SUBAPPLICATION Uebung_087a1 (* Beispiel für E_DEMUX_4 *)
  (* Standard: 61499-2; Description: Copyright (c) 2023 Meisterschulen am Ostbahnhof This program and the accompanying materials are made available under the terms of the Eclipse Public License 2.0 which is available at https://www.eclipse.org/legal/epl-2.0/ SPDX-License-Identifier: EPL-2.0 Beispiel für E_CTD Aufwärts zählen UAO Curriculum Module 3 - The IEC 61499 Standard, Seite 93 *)
  (* Version 1.0, 2023-10-23, Franz Höpfinger, Meisterschulen am Ostbahnhof *)
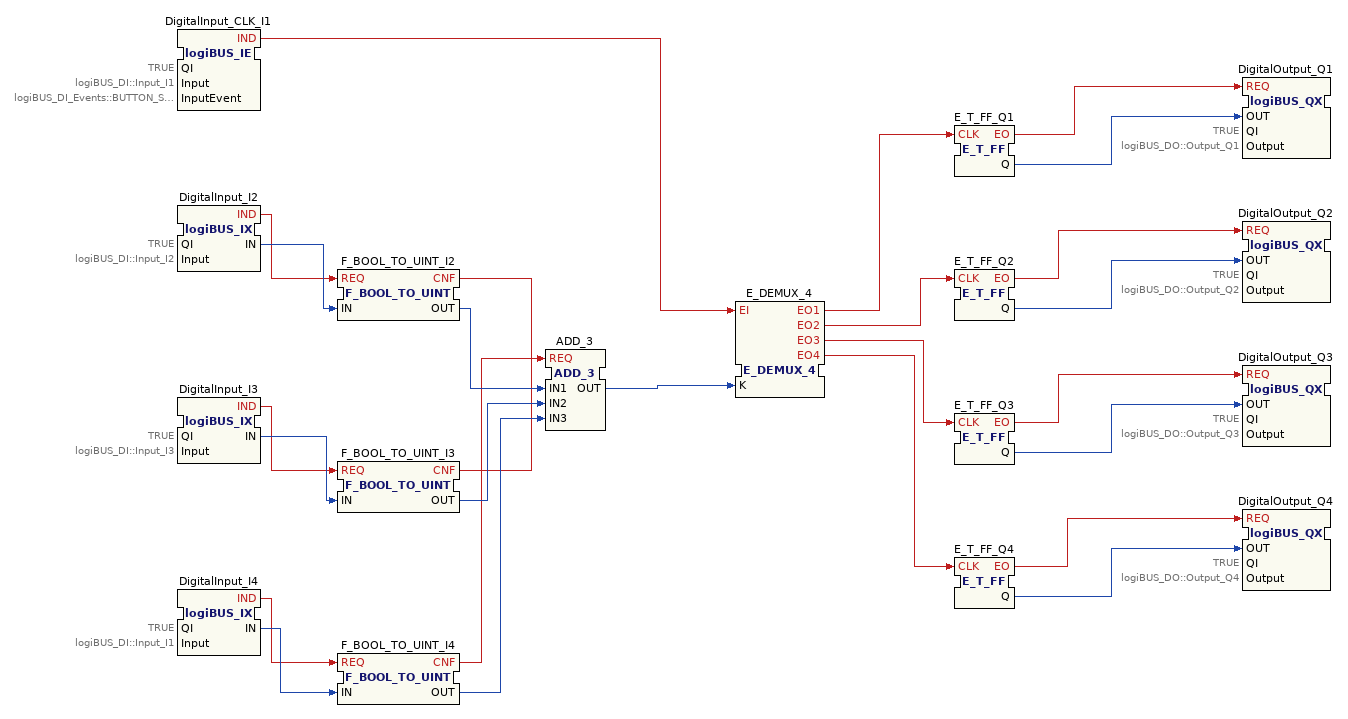
  (* Diese Taste schaltet ein oder aus *)
  (* Die Anzahl der restlichen Tasten bestimmt den Ausgang: Keine --> Q1 Eine --> Q2 Zwei --> Q3 Drei --> Q4 *)
  FBS
    E_DEMUX_4 : E_DEMUX_4;
    ADD_3 : ADD_3;
    DigitalInput_I2 : logiBUS_IX(QI := TRUE, Input := logiBUS_DI::Input_I2);
    DigitalInput_I3 : logiBUS_IX(QI := TRUE, Input := logiBUS_DI::Input_I3);
    DigitalInput_I4 : logiBUS_IX(QI := TRUE, Input := logiBUS_DI::Input_I1);
    F_BOOL_TO_UINT_I2 : F_BOOL_TO_UINT;
    F_BOOL_TO_UINT_I3 : F_BOOL_TO_UINT;
    F_BOOL_TO_UINT_I4 : F_BOOL_TO_UINT;
    DigitalOutput_Q2 : logiBUS_QX(QI := TRUE, Output := logiBUS_DO::Output_Q2);
    DigitalOutput_Q1 : logiBUS_QX(QI := TRUE, Output := logiBUS_DO::Output_Q1);
    DigitalOutput_Q4 : logiBUS_QX(QI := TRUE, Output := logiBUS_DO::Output_Q4);
    DigitalOutput_Q3 : logiBUS_QX(QI := TRUE, Output := logiBUS_DO::Output_Q3);
    E_T_FF_Q1 : E_T_FF;
    E_T_FF_Q2 : E_T_FF;
    E_T_FF_Q3 : E_T_FF;
    E_T_FF_Q4 : E_T_FF;
    DigitalInput_CLK_I1 : logiBUS_IE(QI := TRUE, Input := logiBUS_DI::Input_I1, InputEvent := logiBUS_DI_Events::BUTTON_SINGLE_CLICK);
  END_FBS
  EVENT_CONNECTIONS
    DigitalInput_I2.IND TO F_BOOL_TO_UINT_I2.REQ;
    DigitalInput_I3.IND TO F_BOOL_TO_UINT_I3.REQ;
    DigitalInput_I4.IND TO F_BOOL_TO_UINT_I4.REQ;
    F_BOOL_TO_UINT_I4.CNF TO ADD_3.REQ;
    F_BOOL_TO_UINT_I3.CNF TO ADD_3.REQ;
    F_BOOL_TO_UINT_I2.CNF TO ADD_3.REQ;
    E_T_FF_Q4.EO TO DigitalOutput_Q4.REQ;
    E_T_FF_Q3.EO TO DigitalOutput_Q3.REQ;
    E_T_FF_Q2.EO TO DigitalOutput_Q2.REQ;
    E_T_FF_Q1.EO TO DigitalOutput_Q1.REQ;
    E_DEMUX_4.EO1 TO E_T_FF_Q1.CLK;
    E_DEMUX_4.EO2 TO E_T_FF_Q2.CLK;
    E_DEMUX_4.EO3 TO E_T_FF_Q3.CLK;
    E_DEMUX_4.EO4 TO E_T_FF_Q4.CLK;
    DigitalInput_CLK_I1.IND TO E_DEMUX_4.EI;
  END_CONNECTIONS
  DATA_CONNECTIONS
    DigitalInput_I2.IN TO F_BOOL_TO_UINT_I2.IN;
    DigitalInput_I3.IN TO F_BOOL_TO_UINT_I3.IN;
    DigitalInput_I4.IN TO F_BOOL_TO_UINT_I4.IN;
    F_BOOL_TO_UINT_I2.OUT TO ADD_3.IN1;
    F_BOOL_TO_UINT_I3.OUT TO ADD_3.IN2;
    F_BOOL_TO_UINT_I4.OUT TO ADD_3.IN3;
    ADD_3.OUT TO E_DEMUX_4.K;
    E_T_FF_Q4.Q TO DigitalOutput_Q4.OUT;
    E_T_FF_Q3.Q TO DigitalOutput_Q3.OUT;
    E_T_FF_Q2.Q TO DigitalOutput_Q2.OUT;
    E_T_FF_Q1.Q TO DigitalOutput_Q1.OUT;
  END_CONNECTIONS
END_SUBAPPLICATION
